{attribute addProperty BoxType "KL8528"}
{attribute addProperty Id "Channel_1Channel_9A18274A00"}
{attribute addProperty CRC "3048782480"}
{attribute addProperty SizeInBites "0"}
{attribute addProperty SizeInBytes "0"}
TYPE KL8528_B5B8BA90 :
STRUCT
	{attribute addProperty Name "Channel_1"}
	Channel_1 : Channel_9A18274A;
END_STRUCT
END_TYPE

(* stored: Version 1.2.0.0, ProductVersion 3.1.4024.9
   DUT KL8528_B5B8BA90: Id {fe65998a-eb75-4887-93a6-81c0020a7148} *)
